TYPE ST_MoveRequestStatus :
STRUCT
    bNewMoveReq: BOOL;
    nCmdData: INT;
    nCommand: INT;
	bExecute : BOOL;
    bExecHome: BOOL;
    bExecMove: BOOL;
	bValidatedMove : BOOL;
	bStop : BOOL;
	bReset : BOOL;
	bEnable : BOOL;
	bPrepareDisable : BOOL;
	fPosition:LREAL;
	fVelocity :LREAL;
	fAcceleration :LREAL;
	fDeceleration :LREAL;
	fHomeOffset : LREAL;
END_STRUCT
END_TYPE

(* stored: Version 1.1.0.1
   DUT ST_MoveRequestStatus: Id {a07ca9a6-ee49-49b8-ab2e-03bd2d0e53c7} *)
